FUNCTION_BLOCK StartPauseResetButtons
  (* Standard: 61499-2 *)
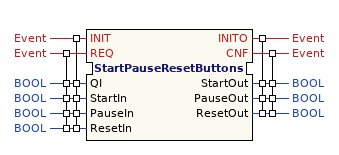
  EVENT_INPUT
    INIT WITH QI, StartIn, PauseIn, ResetIn;
    REQ WITH QI, StartIn, PauseIn, ResetIn;
  END_EVENT
  EVENT_OUTPUT
    INITO WITH StartOut, PauseOut, ResetOut;
    CNF WITH StartOut, PauseOut, ResetOut;
  END_EVENT
  VAR_INPUT
    QI : BOOL;
    StartIn : BOOL;
    PauseIn : BOOL;
    ResetIn : BOOL;
  END_VAR
  VAR_OUTPUT
    StartOut : BOOL;
    PauseOut : BOOL;
    ResetOut : BOOL;
  END_VAR
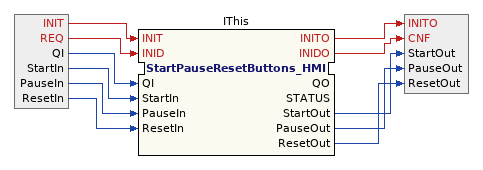
  FBS
    IThis : StartPauseResetButtons_HMI;
  END_FBS
  EVENT_CONNECTIONS
    INIT TO IThis.INIT;
    REQ TO IThis.INID;
    IThis.INITO TO INITO;
    IThis.INIDO TO CNF;
  END_CONNECTIONS
  DATA_CONNECTIONS
    QI TO IThis.QI;
    StartIn TO IThis.StartIn;
    PauseIn TO IThis.PauseIn;
    ResetIn TO IThis.ResetIn;
    IThis.StartOut TO StartOut;
    IThis.PauseOut TO PauseOut;
    IThis.ResetOut TO ResetOut;
  END_CONNECTIONS
END_FUNCTION_BLOCK
